Staubli VAL3: F6_testsync.pgx

program F6_testsync()
begin
  //  if taskStatus("SychMove")==-1
  //    taskCreateSync "SychMove",0.004,bRes,task_sychron()
  //  endIf
end
